// TIA Portal V20 export
DATA_BLOCK "zPMC_Configuration"   // DB357
// stored: MemoryReserve 100, Namespace CITI_Logic
   VAR
      CITI : Array[0..29] of "CITI_Logic.zp_CITI_Configuration";
   END_VAR
BEGIN
END_DATA_BLOCK
